Yaskawa INFORM job: R1-W53NOWA(-180_180).JBI

/JOB
//NAME R1-W53NOWA(-180_180)
//POS
///NPOS 15,15,0,2,0,0
///TOOL 0
///POSTYPE PULSE
///PULSE
C00000=194992,-60991,-78125,34810,68358,6742
C00001=182802,-61941,-57863,34314,60705,57425
C00002=182246,-42212,-43172,34203,61844,57564
C00003=182246,-42148,-42765,34266,61662,57500
C00004=182246,-42212,-43172,34203,61844,57564
C00005=186617,-48203,-47599,25506,55016,63827
C00006=187016,-44944,-45329,23393,56719,68561
C00007=187559,-45791,-45838,23148,56455,68736
C00008=187559,-46401,-50556,22526,58851,69269
C00009=187986,-34014,-47781,18075,78396,62730
C00010=187294,-30584,-44216,18297,78137,62442
C00011=192052,-17346,-34868,16852,78136,64119
C00012=200588,-25504,-60600,13877,87856,68184
C00013=194992,-60991,-78125,34810,68358,6742
C00014=162269,-143776,-121604,48744,43968,-6995
BC00000=361558,70876,1075220
BC00001=361557,70877,1075214
BC00002=361557,70877,1075214
BC00003=361557,70876,1075212
BC00004=361557,70877,1075214
BC00005=361557,70877,1075214
BC00006=361557,70877,1075214
BC00007=361557,70877,1075214
BC00008=361557,70877,1075214
BC00009=361557,70877,1075214
BC00010=361557,70877,1075214
BC00011=361557,70877,1075214
BC00012=361557,66013,1075212
BC00013=361558,70876,1075220
BC00014=361558,70876,1075220
///POSTYPE BASE
///RECTAN
///RCONF 0,0,0,0,1,0,0,0,0,0,0,0,0,0,0,0,0,0,0,0,0,0,0,0
P00006=2.006,1.622,-0.565,0.0000,0.0000,0.0000
P00021=0.073,2.058,-0.109,0.0000,0.0000,0.0000
//INST
///DATE 2023/11/06 18:48
///ATTR SC,RW
///GROUP1 RB1,BS1
NOP
MOVJ C00000 BC00000 VJ=20.00
MOVJ C00001 BC00001 VJ=20.00
MOVL C00002 BC00002 V=60.0
REFP 3 C00003 BC00003
CALL JOB:SEARCH-R1
SET P021 P006
SFTON P021
MOVL C00004 BC00004 V=60.0
MOVL C00005 BC00005 V=60.0
MOVL C00006 BC00006 V=60.0
REFP 3 C00007 BC00007
CALL JOB:SEARCH-R1
SET P021 P006
SFTON P021
MOVL C00008 BC00008 V=60.0
MOVJ C00009 BC00009 VJ=20.00
MACRO1 MJ#(0) ARGF6
SFTON P021
MOVJ C00010 BC00010 VJ=20.00
ARCON
MOVL C00011 BC00011 V=11.7
ARCOF
SFTOF
MOVJ C00012 BC00012 VJ=20.00
MOVJ C00013 BC00013 VJ=20.00
MOVJ C00014 BC00014 VJ=20.00
END
